(* Schneider Machine Expert - Basic project P&N, file version 1.6.0.0 *)
(* ProjectInformations: Name=New project *)

HARDWARE
  Cpu 0: TM221CE16R
  EthernetConfiguration: NetworkName=M221, IpAllocationMode=FixedAddress, IpAddress=0.0.0.0, SubnetMask=0.0.0.0
  SerialLineConfiguration: Baud=Baud19200, Parity=ParityEven, DataBits=DataBits8, StopBits=StopBits1, PhysicalMedium=PhysicalMediumRs485, TransmissionMode=TransmissionModeModbusRtu, SlaveId=1, Addressing=SlaveAddressing
  MastTask: UsePeriodScanMode=false, PeriodScan=100
  FastTask: Period=255
  CpuBehavior: StartingMode=StartAsPreviousState, AutoSaveRamOnEeprom=true, WatchdogPeriod=250

SYMBOLS  (address, symbol, comment, settings)
  %S0       SB_COLDSTART  "Indicates or executes a cold start (data initialized to default values)"
  %S1       SB_WARMSTART  "Indicates there was a warm start with data backup"

POU New POU
  (* SectionNumber=1 *)

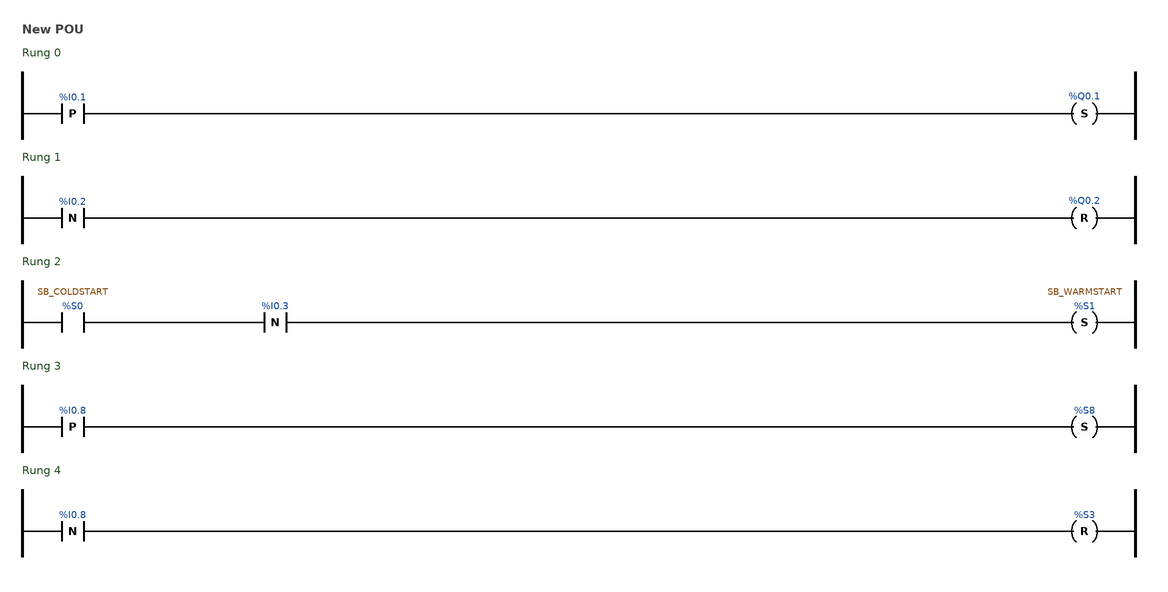

// Rung 0
  LDR %I0.1
  S %Q0.1
  // as ST:
  //   IF RISING(%I0.1) THEN %Q0.1 := TRUE; END_IF;

// Rung 1
  LDF %I0.2
  R %Q0.2
  // as ST:
  //   IF FALLING(%I0.2) THEN %Q0.2 := FALSE; END_IF;

// Rung 2
  LD %S0                  (* SB_COLDSTART *)
  ANDF %I0.3
  S %S1                   (* SB_WARMSTART *)
  // as ST:
  //   IF SB_COLDSTART AND FALLING(%I0.3) THEN SB_WARMSTART := TRUE; END_IF;

// Rung 3
  LDR %I0.8
  S %S8
  // as ST:
  //   IF RISING(%I0.8) THEN %S8 := TRUE; END_IF;

// Rung 4
  LDF %I0.8
  R %S3
  // as ST:
  //   IF FALLING(%I0.8) THEN %S3 := FALSE; END_IF;
